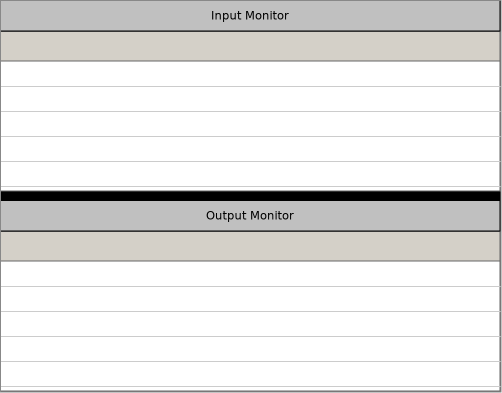
VISUALIZATION IO_Monitor  // 502x393
    Rectangle (0,0 500x391)
    Table (0,31 500x160), data array: InputByte
        p2232123230: Bit7
        p2685023577: InputByte[INDEX]
        p511219082: Bit6
        p1755163831: Bit5
        p4092479075: Bit4
        p2237128397: Bit3
        p505689113: Bit2
        p1757482276: Bit1
        p4088588272: Bit0
        Columns.Column.[3].Template: (InputByte[INDEX].4) <> 0; OnMouseDown: write the text variable via Edit
        Columns.Column.[4].Template: (InputByte[INDEX].3) <> 0; OnMouseDown: write the text variable via Edit
        Columns.Column.[5].Template: (InputByte[INDEX].2) <> 0; OnMouseDown: write the text variable via Edit
        Columns.Column.[0].Template: (InputByte[INDEX].7) <> 0; OnMouseDown: write the text variable via Edit
        Columns.Column.[1].Template: (InputByte[INDEX].6) <> 0; OnMouseDown: write the text variable via Edit
        Columns.Column.[6].Template: (InputByte[INDEX].1) <> 0; OnMouseDown: write the text variable via Edit
        Columns.Column.[2].Template: (InputByte[INDEX].5) <> 0; OnMouseDown: write the text variable via Edit
        Columns.Column.[7].Template: (InputByte[INDEX].0) <> 0; OnMouseDown: write the text variable via Edit
    Rectangle (0,0 500x31), "Input Monitor"
    Table (0,231 500x160), data array: OutputByte
        p2232123230: Bit7
        p511219082: Bit6
        p1755163831: Bit5
        p4092479075: Bit4
        p2237128397: Bit3
        p505689113: Bit2
        p1757482276: Bit1
        p4088588272: Bit0
        Columns.Column.[3].Template: (OutputByte[INDEX].4) <> 0; OnMouseDown: write the text variable via Edit
        Columns.Column.[4].Template: (OutputByte[INDEX].3) <> 0; OnMouseDown: write the text variable via Edit
        Columns.Column.[5].Template: (OutputByte[INDEX].2) <> 0; OnMouseDown: write the text variable via Edit
        Columns.Column.[0].Template: (OutputByte[INDEX].7) <> 0; OnMouseDown: write the text variable via Edit
        Columns.Column.[1].Template: (OutputByte[INDEX].6) <> 0; OnMouseDown: write the text variable via Edit
        Columns.Column.[6].Template: (OutputByte[INDEX].1) <> 0; OnMouseDown: write the text variable via Edit
        Columns.Column.[2].Template: (OutputByte[INDEX].5) <> 0; OnMouseDown: write the text variable via Edit
        Columns.Column.[7].Template: (OutputByte[INDEX].0) <> 0; OnMouseDown: write the text variable via Edit
    Rectangle (0,200 500x31), "Output Monitor"
END_VISUALIZATION

// ---- VISUs/Prog/MANUAL_STEP.TcVIS
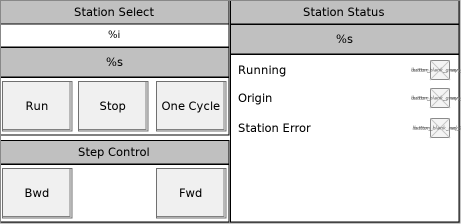
VISUALIZATION MANUAL_STEP  // 461x224
    Rectangle (0,22 229x25), "%i", text variable: Global_Variables_HMI.T_Curr_Step_Station, input disabled if: Global_Variables.M_StepRun
        OnMouseDown: write the text variable via VisuDialogs.Numpad, min 2, max 8
    Rectangle (0,47 229x30), "%s", text variable: Global_Variables_HMI.V_StepRunCurrStation
    Rectangle (0,0 229x24)
    RoundedRectangle (20,-3 188x30), "Station Select"
    Rectangle (0,77 229x58)
    Button (2,81 70x50), "Run"
        tap Global_Variables_HMI.T_StepRun
    Button (78,81 70x50), "Stop"
        tap Global_Variables_HMI.T_StepStop
    Button (156,81 70x50), "One Cycle", pressed state: Global_Variables_HMI.T_OneCycleRun
        toggle Global_Variables_HMI.T_OneCycleRun
    Rectangle (0,140 229x24)
    RoundedRectangle (20,137 188x30), "Step Control"
    Rectangle (0,164 229x58)
    Button (2,168 70x50), "Bwd"
        tap Global_Variables_HMI.T_StepBwd
    Button (156,168 70x50), "Fwd"
        tap Global_Variables_HMI.T_StepFwd
    Rectangle (230,0 229x24)
    RoundedRectangle (250,-3 188x30), "Station Status"
    Rectangle (230,54 229x168)
    RoundedRectangle (235,55 95x30), "Running"
    RoundedRectangle (235,83 95x30), "Origin"
    RoundedRectangle (235,113 95x30), "Station Error"
    Rectangle (230,24 229x30), "%s", text variable: Global_Variables_HMI.V_StepRunStatus
    Frame (430,118 20x20)
        shows Red_Ind(m_Input_Inst := Global_Variables_HMI.T_StationError)
    Frame (430,88 20x20)
        shows Green_Ind(m_Input_Inst := Global_Variables_HMI.T_Origin)
    Frame (430,60 20x20)
        shows Green_Ind(m_Input_Inst := Global_Variables.M_StepRun)
END_VISUALIZATION

// ---- VISUs/Prog/resetbtn.TcVIS
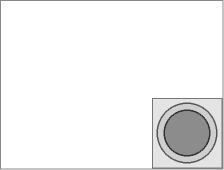
VISUALIZATION resetbtn  // 224x170
    PushSwitch (152,98 70x70), variable: .I_Reset_HMI, behaviour: TAP, style: Switch-PushSwitch-Gray
END_VISUALIZATION

// ---- VISUs/Prog/Std_NewPassWord.TcVIS
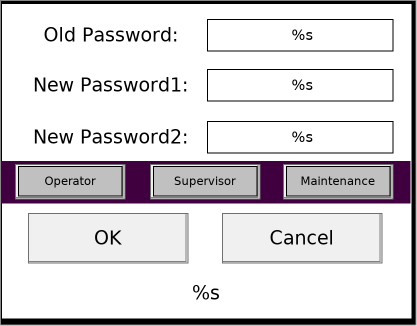
VISUALIZATION Std_NewPassWord  // 417x326
    Group (-2,0 415x322)
        Rectangle (0,0 417x324)
        RoundedRectangle (3,3 411x316)
    RoundedRectangle (17,20 188x30), "Old Password:", invisible if: (In_SelectedPasswordLvl < 2) <> 0
    Rectangle (207,19 186x32), "%s", text variable: Global_Variables_Holding.Password_Control .In_EntryPasswordString, invisible if: (In_SelectedPasswordLvl < 2) <> 0
        OnMouseDown: write the text variable via Edit, min 0, max 10
    Button (28,213 160x50), "OK"
        tap Global_Variables_Holding.Password_Control .In_ChangePassword
    Button (222,213 160x50), "Cancel"
        OnMouseUp: change screen: AssignExpression TP40_SETTING
    RoundedRectangle (9,278 394x30), "%s", text variable: Global_Variables_Holding.Password_Control .Out_StatusString
    RoundedRectangle (17,70 188x30), "New Password1:"
    Rectangle (207,69 186x32), "%s", text variable: Global_Variables_Holding.Password_Control .In_NewPasswordString1
        OnMouseDown: write the text variable via Edit, min 0, max 10
    RoundedRectangle (17,122 188x30), "New Password2:"
    Rectangle (207,121 186x32), "%s", text variable: Global_Variables_Holding.Password_Control .In_NewPasswordString2
        OnMouseDown: write the text variable via Edit, min 0, max 10
    Rectangle (1,161 409x42)
    Button (15,164 110x35), "Operator"
        OnMouseUp: execute { Global_Variables_Holding.Password_Control .In_SelectedPasswordLvl:=(0); }
    Button (150,164 110x35), "Supervisor"
        OnMouseUp: execute { Global_Variables_Holding.Password_Control .In_SelectedPasswordLvl:=(1); }
    Button (283,164 110x35), "Maintenance"
        OnMouseUp: execute { Global_Variables_Holding.Password_Control .In_SelectedPasswordLvl:=(2); }
    RoundedRectangle (18,166 104x30), "Operator", colour toggle: Global_Variables_Holding.Password_Control .In_SelectedPasswordLvl = 0
        OnMouseUp: execute { Global_Variables_Holding.Password_Control .In_SelectedPasswordLvl:=(0); }
    RoundedRectangle (153,166 104x30), "Supervisor", colour toggle: Global_Variables_Holding.Password_Control .In_SelectedPasswordLvl = 1
        OnMouseUp: execute { Global_Variables_Holding.Password_Control .In_SelectedPasswordLvl:=(1); }
    RoundedRectangle (286,166 104x30), "Maintenance", colour toggle: Global_Variables_Holding.Password_Control .In_SelectedPasswordLvl = 2
        OnMouseUp: execute { Global_Variables_Holding.Password_Control .In_SelectedPasswordLvl:=(2); }
END_VISUALIZATION

// ---- VISUs/Prog/Std_Password.TcVIS
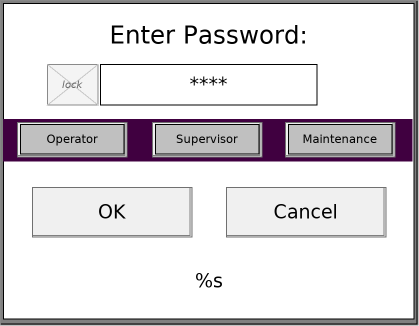
VISUALIZATION Std_Password  // 419x326
    Group (0,0 415x322)
        Rectangle (0,0 417x324)
        RoundedRectangle (3,3 411x316)
    Rectangle (3,119 409x42)
    RoundedRectangle (89,20 240x30), "Enter Password:"
    Rectangle (100,64 217x41), "****", text variable: Global_Variables_Holding.Password_Control .In_EntryPasswordString
        OnMouseDown: write the text variable via Edit, min 0, max 10, password
    Button (32,187 160x50), "OK"
        tap Global_Variables_Holding.Password_Control .In_EnterPassword
    Button (226,187 160x50), "Cancel"
        OnMouseUp: change screen: AssignExpression TP00_MAIN
    RoundedRectangle (89,266 240x30), "%s", text variable: Global_Variables_Holding.Password_Control .Out_StatusString
    Image (47,64 51x41), image: lock
    Button (17,122 110x35), "Operator"
        OnMouseUp: execute { Global_Variables_Holding.Password_Control .In_SelectedPasswordLvl:=(0); }
    Button (152,122 110x35), "Supervisor"
        OnMouseUp: execute { Global_Variables_Holding.Password_Control .In_SelectedPasswordLvl:=(1); }
    Button (285,122 110x35), "Maintenance"
        OnMouseUp: execute { Global_Variables_Holding.Password_Control .In_SelectedPasswordLvl:=(2); }
    RoundedRectangle (20,124 104x30), "Operator", colour toggle: Global_Variables_Holding.Password_Control .In_SelectedPasswordLvl = 0
        OnMouseUp: execute { Global_Variables_Holding.Password_Control .In_SelectedPasswordLvl:=(0); }
    RoundedRectangle (155,124 104x30), "Supervisor", colour toggle: Global_Variables_Holding.Password_Control .In_SelectedPasswordLvl = 1
        OnMouseUp: execute { Global_Variables_Holding.Password_Control .In_SelectedPasswordLvl:=(1); }
    RoundedRectangle (288,124 104x30), "Maintenance", colour toggle: Global_Variables_Holding.Password_Control .In_SelectedPasswordLvl = 2
        OnMouseUp: execute { Global_Variables_Holding.Password_Control .In_SelectedPasswordLvl:=(2); }
END_VISUALIZATION
